(* PLC project Unnamed, Unknown Unnamed 1 *)
(* stored: creationDateTime 2022-05-06T11:12:02, modificationDateTime 2022-05-09T09:09:01 *)

PROGRAM program0
  VAR
    trendval0 : HMI_REAL;
    trendval1 : HMI_REAL;
    counter : INT;
  END_VAR
  VAR  (* added by the conversion: wires and edge detectors of the diagram *)
    _ADD4_OUT : INT;
    _SEL5_OUT : INT;
    _DIV14_OUT : REAL;
  END_VAR

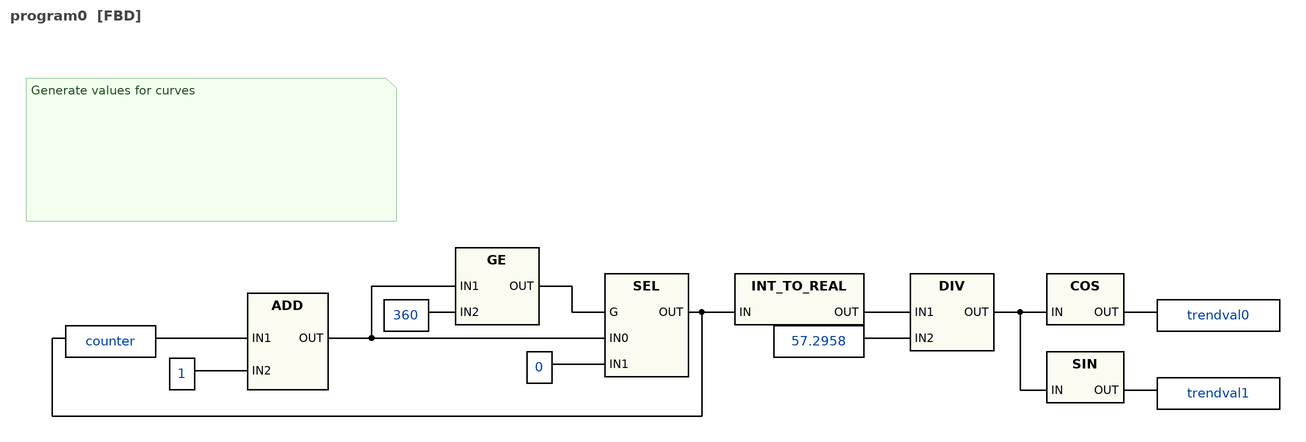
(* FBD diagram, written out as Structured Text *)
(* Generate values for curves *)
_ADD4_OUT := counter + 1;
_SEL5_OUT := SEL(_ADD4_OUT >= 360, _ADD4_OUT, 0);
_DIV14_OUT := INT_TO_REAL(_SEL5_OUT) / 57.2958;
trendval0 := COS(_DIV14_OUT);
counter := _SEL5_OUT;
trendval1 := SIN(_DIV14_OUT);
END_PROGRAM

CONFIGURATION config
  RESOURCE resource1 ON PLC
    TASK task0(INTERVAL := T#20ms, PRIORITY := 0);
    PROGRAM instance0 WITH task0 : program0;
  END_RESOURCE
END_CONFIGURATION
